FUNCTION_BLOCK PUBLIC FB_Observer IMPLEMENTS I_Observer
VAR
	fValue				: LREAL;
END_VAR

{attribute 'monitoring':='call'}
PROPERTY PUBLIC fActualValue : LREAL
GET
fActualValue := THIS^.fValue;
END_GET
END_PROPERTY

METHOD PUBLIC Update
VAR_INPUT
	fValue			: LREAL;
END_VAR
THIS^.fValue := fValue;
END_METHOD

END_FUNCTION_BLOCK

(* stored: Version 1.1.0.1, ProductVersion 3.1.4022.10
   POU FB_Observer: Id {c2f07dc9-2028-42d5-bdcb-a6253ab74410}, SpecialFunc None
   Property fActualValue: Id {f671e0f9-25f6-47ac-a38a-ee6697f9367c}
   Get Get: Id {4ec82d87-f4c6-4d3d-bfce-1210b040861c}
   Method Update: Id {a3fc2fe7-b922-4dd5-aa75-b531f9951d99} *)
